Staubli VAL3: onF5Event.pgx

program onF5Event()
begin
end
